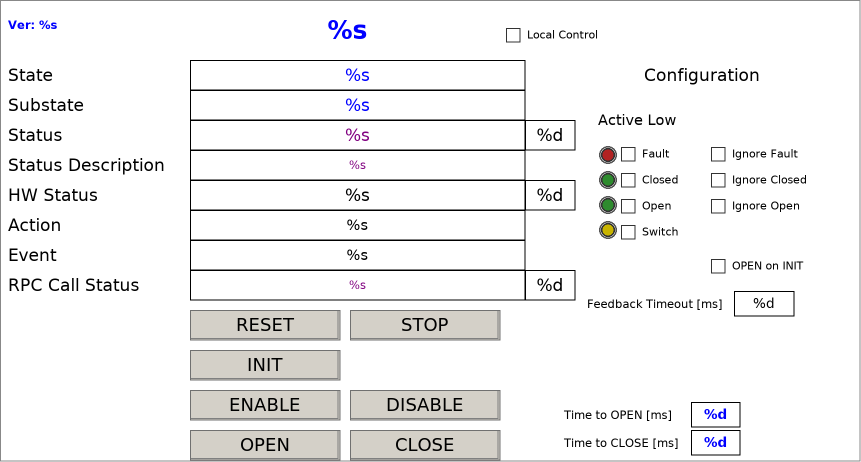
VISUALIZATION GUI_TEMPLATE_SHUTTER  // 861x462
VAR_IN_OUT
	m_Instance:	FB_SHUTTER;
END_VAR
    Rectangle (190,60 335x30), "%s", text variable: m_Instance.stat.sState
    Rectangle (190,90 335x30), "%s", text variable: m_Instance.stat.sSubstate
    Button (190,310 150x30), "RESET", input disabled if: (m_Instance.stat.bLocal = FALSE) <> 0
        OnMouseDown: execute { m_Instance.ctrl.nCommand :=E_SHUTTER_COMMAND.RESET; m_Instance.ctrl.bExecute := TRUE; }
    Button (190,350 150x30), "INIT", input disabled if: (m_Instance.stat.bLocal = FALSE) <> 0
        OnMouseDown: execute { m_Instance.ctrl.nCommand := E_SHUTTER_COMMAND.INIT; m_Instance.ctrl.bExecute := TRUE; }
    Button (350,310 150x30), "STOP", input disabled if: (m_Instance.stat.bLocal = FALSE) <> 0
        OnMouseDown: execute { m_Instance.ctrl.nCommand := E_SHUTTER_COMMAND.STOP; m_Instance.ctrl.bExecute := TRUE; }
    Button (190,390 150x30), "ENABLE", input disabled if: (m_Instance.stat.bLocal = FALSE) <> 0
        OnMouseDown: execute { m_Instance.ctrl.nCommand := E_SHUTTER_COMMAND.ENABLE; m_Instance.ctrl.bExecute := TRUE; }
    Button (350,390 150x30), "DISABLE", input disabled if: (m_Instance.stat.bLocal = FALSE) <> 0
        OnMouseDown: execute { m_Instance.ctrl.nCommand := E_SHUTTER_COMMAND.DISABLE; m_Instance.ctrl.bExecute := TRUE; }
    Button (190,430 150x30), "OPEN", input disabled if: (m_Instance.stat.bLocal = FALSE) <> 0
        OnMouseDown: execute { m_Instance.ctrl.nCommand := E_SHUTTER_COMMAND.OPEN; m_Instance.ctrl.bExecute := TRUE; }
    Button (350,430 150x30), "CLOSE", input disabled if: (m_Instance.stat.bLocal = FALSE) <> 0
        OnMouseDown: execute { m_Instance.ctrl.nCommand := E_SHUTTER_COMMAND.CLOSE; m_Instance.ctrl.bExecute := TRUE; }
    Rectangle (5,60 180x30), "State"
    Rectangle (5,90 180x30), "Substate"
    Rectangle (190,120 335x30), "%s", text variable: m_Instance.stat.sStatus
    Rectangle (190,150 335x30), "%s", text variable: m_Instance.stat.sErrorText
    Rectangle (5,120 180x30), "Status"
    Rectangle (5,150 180x30), "Status Description"
    Rectangle (190,210 335x30), "%s", text variable: m_Instance.stat.sActionDesc
    Rectangle (190,240 335x30), "%s", text variable: m_Instance.stat.sEventDesc
    Rectangle (190,180 335x30), "%s", text variable: m_Instance.stat.sHwStatus
    Rectangle (5,180 180x30), "HW Status"
    Rectangle (525,180 50x30), "%d", text variable: m_Instance.stat.nHwStatus
    Rectangle (5,210 180x30), "Action"
    Rectangle (5,240 180x30), "Event"
    Rectangle (190,12 315x35), "%s", text variable: m_Instance.cfg.sName
    Rectangle (525,120 50x30), "%d", text variable: m_Instance.stat.nStatus
    Checkbox (504,20 116x30), "Local Control", variable: m_Instance.stat.bLocal
    Rectangle (641,60 180x30), "Configuration"
    Rectangle (595,105 126x30), "Active Low"
    Checkbox (619,139 75x30), "Fault", variable: m_Instance.cfg.bActiveLowFault, input disabled if: (m_Instance.stat.bLocal = FALSE) <> 0
    Checkbox (709,139 110x30), "Ignore Fault", variable: m_Instance.cfg.bIgnoreFault, input disabled if: (m_Instance.stat.bLocal = FALSE) <> 0
    Checkbox (619,165 75x30), "Closed", variable: m_Instance.cfg.bActiveLowClosed, input disabled if: (m_Instance.stat.bLocal = FALSE) <> 0
    Checkbox (619,217 75x30), "Switch", variable: m_Instance.cfg.bActiveLowSwitch, input disabled if: (m_Instance.stat.bLocal = FALSE) <> 0
    Checkbox (709,251 150x30), "OPEN on INIT", tooltip "If selected, the default state of the shutter on INIT or DISABLE will be OPEN.", variable: m_Instance.cfg.bInitialState, input disabled if: (m_Instance.stat.bLocal = FALSE) <> 0
    Rectangle (734,291 60x25), "%d", tooltip "When controlling shutter, feedback signal should change within this period.", text variable: m_Instance.cfg.nTimeout, input disabled if: (m_Instance.stat.bLocal = FALSE) <> 0
        OnMouseDown: write the text variable via Default, min 0
    Rectangle (584,294 146x20), "Feedback Timeout [ms]"
    Checkbox (619,191 75x30), "Open", variable: m_Instance.cfg.bActiveLowOpen, input disabled if: (m_Instance.stat.bLocal = FALSE) <> 0
    Checkbox (709,165 110x30), "Ignore Closed", variable: m_Instance.cfg.bIgnoreClosed, input disabled if: (m_Instance.stat.bLocal = FALSE) <> 0
    Checkbox (709,191 110x30), "Ignore Open", variable: m_Instance.cfg.bIgnoreOpen, input disabled if: (m_Instance.stat.bLocal = FALSE) <> 0
    Rectangle (190,270 335x30), "%s", text variable: m_Instance.stat.sRPCErrorText
    Rectangle (5,270 180x30), "RPC Call Status"
    Rectangle (5,10 99x30), "Ver: %s", tooltip "'Shutter.library version'", text variable: m_Instance.stat.sLibVersion, input disabled if: true
    Rectangle (561,405 124x20), "Time to OPEN [ms]"
    Rectangle (561,433 124x20), "Time to CLOSE [ms]"
    Rectangle (691,402 49x25), "%d", tooltip "Last opening time [ms]. -1 means not open yet.", text variable: m_Instance.stat.nLastTimeToOpen
    Rectangle (691,430 49x25), "%d", tooltip "Last closing time [ms]. -1 means not closed yet.", text variable: m_Instance.stat.nLastTimeToClose
    Rectangle (525,270 50x30), "%d", tooltip "RPC Error Code 0 - OK", text variable: m_Instance.stat.nRpcErrorCode
    Lamp1 (598,145 20x20), tooltip "If ON, Fault signal is active.", variable: m_Instance.bFault, style: Lamp-Lamp1-Red
    Lamp1 (598,170 20x20), tooltip "If ON, Closed signal is active.", variable: m_Instance.bClosed, style: Lamp-Lamp1-Green
    Lamp1 (598,195 20x20), tooltip "If ON, Open signal is active.", variable: m_Instance.bOpen, style: Lamp-Lamp1-Green
    Lamp1 (598,220 20x20), tooltip "If ON, digital control output is high.", variable: m_Instance.q_bSwitch, style: Lamp-Lamp1-Yellow
END_VISUALIZATION

(* stored: Version 1.1.0.1, ProductVersion 3.1.4022.16
   Visu GUI_TEMPLATE_SHUTTER: Id {208abcb1-f1a3-4a00-92a5-f362cd7556ac} *)
